(* CODESYS project DataStreams.project

Project tree, tasks and I/O mapping:
  Device : CODESYS Control Win V3, 3S - Smart Software Solutions GmbH, version 3.5.12.30
    application Application
      libraries: Standard, * (System); BASIC, 3.3.3.0 (OSCAT); BR_MQTTClient, 1.2.0.1 (Bedrock Automation)
      task MainTask (cyclic, interval 4 ms, priority 1) calls Timers, DataStreams, Randomiser, ID_Constructor, Machine_State_Handler
      task Pick_and_Place (cyclic, interval 5000 ms, priority 1) calls Pick_and_Place
      task TankControl (cyclic, interval t#20ms, priority 1) calls _Main
      global variables GVL
      Symbols
      DUT/
        data type DS_Angle
        data type DS_BlockWave
        data type DS_Sys_Info
        data type DS_MachineState
        data type DS_Machine_Info
        data type DUT_ControlValve
        data type DUT_Motor
        data type DUT_StorageTank
        data type DUT_Switch
        data type DUT_Transmitter
        data type DUT_Valve
      POU/
        program Timers [LD]
        program DataStreams [ST]
        program Randomiser [CFC]
        program ID_Constructor [ST]
        program Pick_and_Place [ST]
        program Machine_State_Handler [LD]
        program MQTT_Client [CFC]
        program AgitatorControl [ST]
        program LevelControl [ST]
        program PumpControl [ST]
        program ValveControl [LD]
        program _Main [ST]
    Ethernet : Ethernet, 3S - Smart Software Solutions GmbH, version 3.5.11.0
        settings: IPAddress = [172,31,33,236]; SubnetMask = [255,255,240,0]; GatewayAddress = [172,31,32,1]; MACAddress = [16#0E,16#C7,16#4C,16#B6,16#0D,16#8C]; NetworkInterfaceName = 'Ethernet'; NetworkInterfaceName = "Ethernet"; SaveCommunicationSettings = FALSE
      ModbusTCP_Slave_Device : ModbusTCP Slave Device, 3S - Smart Software Solutions GmbH, version 3.5.12.0
          output Application.Machine_State.Start : BOOL  // Outputs.Outputs.Bit0
          output Application.Machine_State.Stop : BOOL  // Outputs.Outputs.Bit1
          output Application.Machine_State.Mode : WORD  // Outputs.Outputs
          output Application.Machine_State.State : WORD  // Outputs.Outputs
          unmapped channels: Inputs, Outputs
*)

// Device/Application/DUT/DS_Angle
TYPE DS_Angle :
STRUCT
     Angle : REAL;
     Sine  : LREAL;
END_STRUCT
END_TYPE

// Device/Application/DUT/DS_BlockWave
TYPE DS_BlockWave :
STRUCT
	Number_of_Waves : SINT;
	Amplitude  : LREAL;
END_STRUCT
END_TYPE

// Device/Application/DUT/DS_Sys_Info
TYPE DS_Sys_Info :
STRUCT
    CPU_Usage : UDINT;
    SYS_Latency : UDINT;
	SYS_Latency_max : UDINT;
END_STRUCT
END_TYPE

// Device/Application/DUT/DS_MachineState
TYPE DS_MachineState :
STRUCT
	Mode	: WORD:=1;
	State   : WORD:=0;
	Start	: BOOL:=0;
	Stop	: BOOL:=0;
END_STRUCT
END_TYPE

// Device/Application/DUT/DS_Machine_Info
TYPE DS_Machine_Info :
STRUCT
	Item_ID 		: STRING;
	Move_result		: STRING;
	Motor_current	: REAL;
END_STRUCT
END_TYPE

// Device/Application/DUT/DUT_ControlValve
TYPE DUT_ControlValve :
STRUCT
	FB_Position: REAL;
	Request: REAL;
END_STRUCT
END_TYPE

// Device/Application/DUT/DUT_Motor
TYPE DUT_Motor :
STRUCT
	FB_Running:BOOL;
	Request:BOOL;
END_STRUCT
END_TYPE

// Device/Application/DUT/DUT_StorageTank
TYPE DUT_StorageTank :
STRUCT
	FeedValve_A: DUT_Valve;
	FeedValve_B: DUT_Valve;
	FeedValve_C: DUT_Valve;
	Agitator: DUT_Motor;
	Pump: DUT_Motor;
	Tank_HLS: DUT_Switch;
	Tank_LLS: DUT_Switch;
	Tank_LT: DUT_Transmitter;
	Tank_TT: DUT_Transmitter;
	Tank_CV: DUT_ControlValve;
    Pipe_PT: DUT_Transmitter;	
END_STRUCT
END_TYPE

// Device/Application/DUT/DUT_Switch
TYPE DUT_Switch :
STRUCT
	FB_Activated:BOOL;
END_STRUCT
END_TYPE

// Device/Application/DUT/DUT_Transmitter
TYPE DUT_Transmitter :
STRUCT
	FB_Value: REAL;
END_STRUCT
END_TYPE

// Device/Application/DUT/DUT_Valve
TYPE DUT_Valve :
STRUCT
   FB_Open: BOOL:=FALSE;
   FB_Closed: BOOL:=TRUE;
   Request: BOOL:=FALSE;
END_STRUCT
END_TYPE

// Device/Application/GVL
VAR_GLOBAL
    Always_On: BOOL := 1;
    T1s: BOOL;
    T5s: BOOL;
    T100ms: BOOL;

    Data_Streams: ARRAY[0..2] OF DS_Angle;
	Temp_Item_ID : STRING[9] := 'AWS-     ';
	Temp_Item_ID_Pos : SINT := 4;
	System_Info: DS_Sys_Info;
	BlockWave: DS_BlockWave;

	Random_Number: REAL;
	Random_Character: STRING;
	Random_TrueFalse: REAL;
	
	Machine_Info: DS_Machine_Info;
	Machine_State: DS_MachineState;
	
	StorageTank: DUT_StorageTank;
    
END_VAR

// Device/Application/POU/Timers
PROGRAM Timers
VAR
	TON_5s: TON;
	TON_1s: TON;
	TON_100ms: TON;
END_VAR

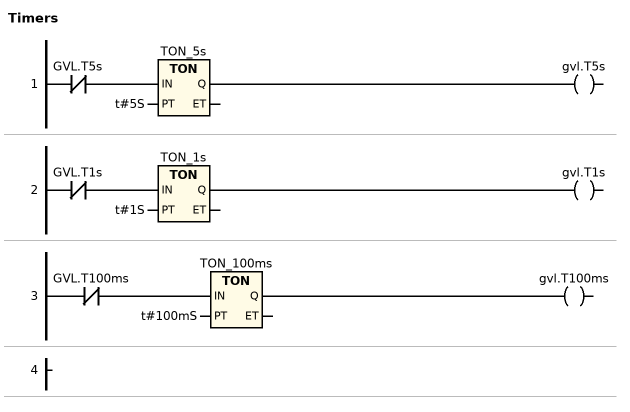
// NETWORK 1
TON_5s(IN := NOT GVL.T5s, PT := t#5S); // TON
gvl.T5s := TON_5s.Q;

// NETWORK 2
TON_1s(IN := NOT GVL.T1s, PT := t#1S); // TON
gvl.T1s := TON_1s.Q;

// NETWORK 3
TON_100ms(IN := NOT GVL.T100ms, PT := t#100mS); // TON
gvl.T100ms := TON_100ms.Q;

// NETWORK 4

END_PROGRAM

// Device/Application/POU/DataStreams
PROGRAM DataStreams
VAR
  iCounter: SINT;
	
	iSin: REAL;
END_VAR

IF gvl.T100ms THEN
	gvl.Data_Streams[0].Angle := gvl.Data_Streams[0].Angle + 0.1; 
	IF gvl.Data_Streams[0].Angle > 180 THEN 
		gvl.Data_Streams[0].Angle := -179.9;	
	END_IF
	gvl.Data_Streams[0].Sine :=  180* (SIN((gvl.Data_Streams[0].Angle * 3.14159265359)/180));
    IF gvl.Machine_State.State=1 THEN gvl.Machine_Info.Motor_current:=gvl.Machine_Info.Motor_current+0.2;END_IF
	IF gvl.Machine_Info.Motor_current>=5 THEN gvl.Machine_Info.Motor_current:=4.8; END_IF
	IF gvl.Machine_State.State=3 THEN gvl.Machine_Info.Motor_current:=gvl.Machine_Info.Motor_current-0.05; END_IF
    gvl.BlockWave.Amplitude:=0;
    iCounter:=1;
    WHILE iCounter <= gvl.BlockWave.Number_of_Waves DO 
        iSin :=(180* (SIN((gvl.Data_Streams[0].Angle * 3.14159265359 * iCounter)/180)))/iCounter;
        gvl.BlockWave.Amplitude:=gvl.BlockWave.Amplitude + iSin ;	
		iCounter:=iCounter+2;
    END_WHILE;
END_IF

IF gvl.T1s THEN
	gvl.Data_Streams[1].Angle := gvl.Data_Streams[1].Angle + 1; 
	IF gvl.Data_Streams[1].Angle > 180 THEN 
		gvl.Data_Streams[1].Angle := -179;	
	END_IF
	gvl.Data_Streams[1].Sine := 180* (SIN((gvl.Data_Streams[1].Angle * 3.14159265359)/180)); 
END_IF

IF gvl.T5s THEN
	gvl.Data_Streams[2].Angle := gvl.Data_Streams[2].Angle + 5; 
	IF gvl.Data_Streams[2].Angle > 180 THEN 
		gvl.Data_Streams[2].Angle := -175;	
	END_IF
	gvl.Data_Streams[2].Sine := 180* (SIN((gvl.Data_Streams[2].Angle * 3.14159265359)/180)); 
END_IF

IF gvl.Machine_State.State=0 THEN gvl.Machine_Info.Motor_current:=0; END_IF;
IF gvl.Machine_State.State=2 THEN gvl.Machine_Info.Motor_current:=5; END_IF

END_PROGRAM

// Device/Application/POU/Randomiser
PROGRAM Randomiser
VAR
END_VAR
VAR // added by the converter: edge detectors and wires of the graphical bodies
    _w1, _w2, _w3, _w4 : ANY;
END_VAR

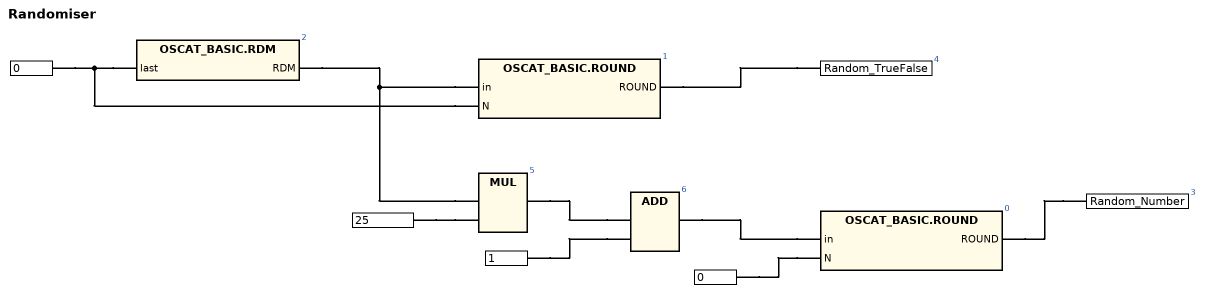
_w2 := OSCAT_BASIC.ROUND(in := _w1, N := 0);
_w4 := OSCAT_BASIC.ROUND(in := _w3, N := 0);
_w3 := OSCAT_BASIC.RDM(last := 0);
Random_Number := _w2;
Random_TrueFalse := _w4;
_w1 := _w3 * 25 + 1;

END_PROGRAM

// Device/Application/POU/ID_Constructor
PROGRAM ID_Constructor
VAR
	Identity:STRING[4];
	ASCII_Code:SINT;	
END_VAR

ASCII_Code:=REAL_TO_SINT(gvl.Random_Number)+64;
gvl.Temp_Item_ID[gvl.Temp_Item_ID_Pos]:=ASCII_Code;
gvl.Temp_Item_ID_Pos:=gvl.Temp_Item_ID_Pos+1;
IF gvl.Temp_Item_ID_Pos=9 THEN gvl.Temp_Item_ID_Pos:=4; END_IF;

END_PROGRAM

// Device/Application/POU/Machine_State_Handler
PROGRAM Machine_State_Handler
VAR
	Stopped:BOOL:=TRUE;
	Starting:BOOL;
	Started:BOOL;
	Stopping:BOOL;	
	TON_0: TON;
	TON_1: TON;
END_VAR
VAR // added by the converter: edge detectors and wires of the graphical bodies
    _w1, _w2, _w3, _w4 : BOOL;
END_VAR

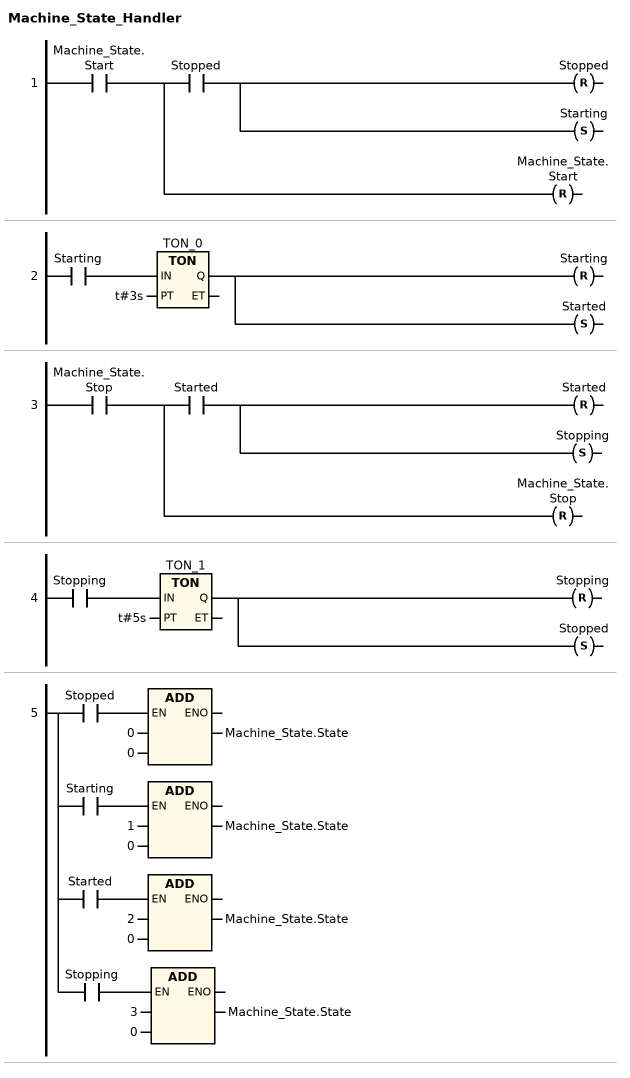
// NETWORK 1
_w1 := Machine_State.Start;
_w2 := _w1 AND Stopped;
Stopped R= _w2;
Starting S= _w2;
Machine_State.Start R= _w1;

// NETWORK 2
TON_0(IN := Starting, PT := t#3s); // TON
Starting R= TON_0.Q;
Started S= TON_0.Q;

// NETWORK 3
_w3 := Machine_State.Stop;
_w4 := _w3 AND Started;
Started R= _w4;
Stopping S= _w4;
Machine_State.Stop R= _w3;

// NETWORK 4
TON_1(IN := Stopping, PT := t#5s); // TON
Stopping R= TON_1.Q;
Stopped S= TON_1.Q;

// NETWORK 5
IF Stopped THEN Machine_State.State := 0 + 0; END_IF
IF Starting THEN Machine_State.State := 1 + 0; END_IF
IF Started THEN Machine_State.State := 2 + 0; END_IF
IF Stopping THEN Machine_State.State := 3 + 0; END_IF

END_PROGRAM

// Device/Application/POU/Pick_and_Place
PROGRAM Pick_and_Place
VAR
END_VAR

IF gvl.Machine_state.State=2 THEN
	gvl.Machine_Info.Item_ID:=gvl.Temp_Item_ID;	
	IF gvl.Random_TrueFalse=1 THEN gvl.Machine_Info.Move_result:='Succes'; ELSE gvl.Machine_Info.Move_result:='Rejected';	
	END_IF
END_IF

END_PROGRAM

// Device/Application/POU/_Main
PROGRAM _Main
VAR
END_VAR

AgitatorControl();
LevelControl();
PumpControl();
ValveControl();

END_PROGRAM

// Device/Application/POU/AgitatorControl
PROGRAM AgitatorControl
VAR
END_VAR

gvl.StorageTank.Agitator.FB_Running:=gvl.StorageTank.Agitator.Request;

END_PROGRAM

// Device/Application/POU/LevelControl
PROGRAM LevelControl
VAR
END_VAR

IF (gvl.StorageTank.FeedValve_A.FB_Open OR gvl.StorageTank.FeedValve_B.FB_Open OR gvl.StorageTank.FeedValve_C.FB_Open) AND gvl.T100ms AND gvl.StorageTank.Tank_LT.FB_Value<100
THEN
	gvl.StorageTank.Tank_LT.FB_Value:=gvl.StorageTank.Tank_LT.FB_Value+0.5;
END_IF

IF gvl.StorageTank.Tank_LT.FB_Value>=100 
THEN 
    gvl.StorageTank.Tank_LT.FB_Value:=100;
	gvl.StorageTank.Tank_HLS.FB_Activated:=TRUE;
ELSE
	gvl.StorageTank.Tank_HLS.FB_Activated:=FALSE;
END_IF

IF gvl.StorageTank.Pump.FB_Running AND gvl.StorageTank.Tank_LT.FB_Value>0 AND gvl.T100ms
THEN
	gvl.StorageTank.Tank_LT.FB_Value:=gvl.StorageTank.Tank_LT.FB_Value-0.25;
END_IF

IF gvl.StorageTank.Tank_LT.FB_Value<=0 
THEN
    gvl.StorageTank.Tank_LT.FB_Value:=0;
	IF gvl.T5s THEN gvl.StorageTank.Tank_LLS.FB_Activated:=TRUE; END_IF
ELSE
	gvl.StorageTank.Tank_LLS.FB_Activated:=FALSE;
END_IF

END_PROGRAM

// Device/Application/POU/PumpControl
PROGRAM PumpControl
VAR
END_VAR

IF NOT(gvl.StorageTank.Tank_LLS.FB_Activated)
THEN
    gvl.StorageTank.Pump.FB_Running:=gvl.StorageTank.Pump.Request;
ELSE
	gvl.StorageTank.Pump.FB_Running:=FALSE;
END_IF

END_PROGRAM

// Device/Application/POU/ValveControl
PROGRAM ValveControl
VAR
	TON_0: TON;
	TON_1: TON;
	TON_3: TON;
	TON_4: TON;
	TON_5: TON;
	TON_6: TON;
END_VAR
VAR // added by the converter: edge detectors and wires of the graphical bodies
    _w1, _w2, _w3, _w4, _w5, _w6 : BOOL;
END_VAR

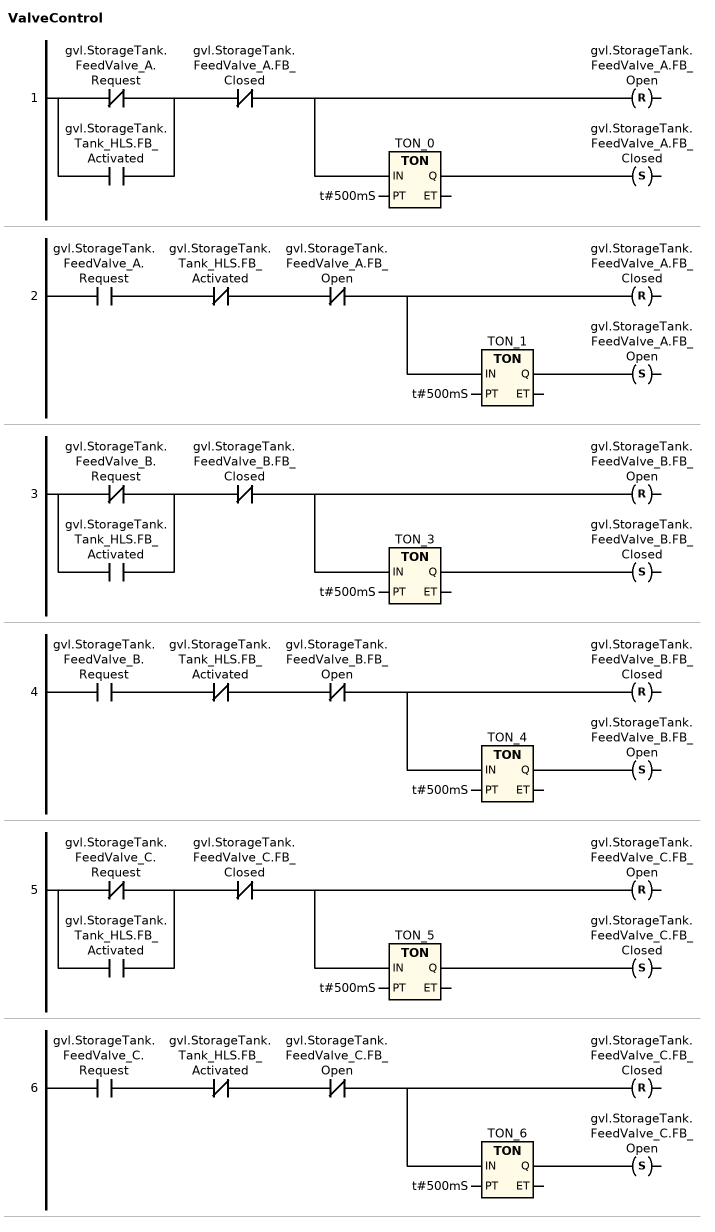
// NETWORK 1
_w1 := (NOT gvl.StorageTank.FeedValve_A.Request OR gvl.StorageTank.Tank_HLS.FB_Activated) AND NOT gvl.StorageTank.FeedValve_A.FB_Closed;
gvl.StorageTank.FeedValve_A.FB_Open R= _w1;
TON_0(IN := _w1, PT := t#500mS); // TON
gvl.StorageTank.FeedValve_A.FB_Closed S= TON_0.Q;

// NETWORK 2
_w2 := gvl.StorageTank.FeedValve_A.Request AND NOT gvl.StorageTank.Tank_HLS.FB_Activated AND NOT gvl.StorageTank.FeedValve_A.FB_Open;
gvl.StorageTank.FeedValve_A.FB_Closed R= _w2;
TON_1(IN := _w2, PT := t#500mS); // TON
gvl.StorageTank.FeedValve_A.FB_Open S= TON_1.Q;

// NETWORK 3
_w3 := (NOT gvl.StorageTank.FeedValve_B.Request OR gvl.StorageTank.Tank_HLS.FB_Activated) AND NOT gvl.StorageTank.FeedValve_B.FB_Closed;
gvl.StorageTank.FeedValve_B.FB_Open R= _w3;
TON_3(IN := _w3, PT := t#500mS); // TON
gvl.StorageTank.FeedValve_B.FB_Closed S= TON_3.Q;

// NETWORK 4
_w4 := gvl.StorageTank.FeedValve_B.Request AND NOT gvl.StorageTank.Tank_HLS.FB_Activated AND NOT gvl.StorageTank.FeedValve_B.FB_Open;
gvl.StorageTank.FeedValve_B.FB_Closed R= _w4;
TON_4(IN := _w4, PT := t#500mS); // TON
gvl.StorageTank.FeedValve_B.FB_Open S= TON_4.Q;

// NETWORK 5
_w5 := (NOT gvl.StorageTank.FeedValve_C.Request OR gvl.StorageTank.Tank_HLS.FB_Activated) AND NOT gvl.StorageTank.FeedValve_C.FB_Closed;
gvl.StorageTank.FeedValve_C.FB_Open R= _w5;
TON_5(IN := _w5, PT := t#500mS); // TON
gvl.StorageTank.FeedValve_C.FB_Closed S= TON_5.Q;

// NETWORK 6
_w6 := gvl.StorageTank.FeedValve_C.Request AND NOT gvl.StorageTank.Tank_HLS.FB_Activated AND NOT gvl.StorageTank.FeedValve_C.FB_Open;
gvl.StorageTank.FeedValve_C.FB_Closed R= _w6;
TON_6(IN := _w6, PT := t#500mS); // TON
gvl.StorageTank.FeedValve_C.FB_Open S= TON_6.Q;

END_PROGRAM

// Device/Application/POU/MQTT_Client
PROGRAM MQTT_Client
VAR
	MQTT_Client1: BR_MQTTClient;
END_VAR

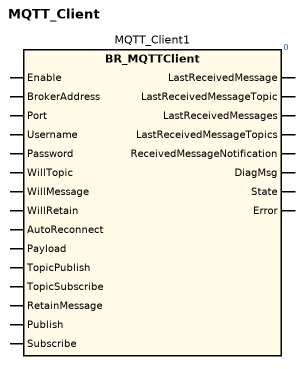
MQTT_Client1(); // BR_MQTTClient

END_PROGRAM
